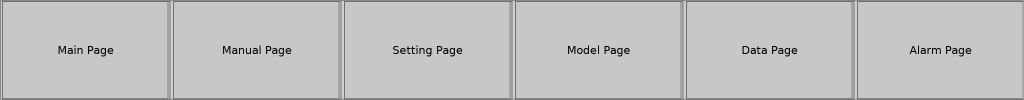
VISUALIZATION LowerBar  // 1024x100
    Button (2,1 168x99), "Main Page", colour toggle: gvl_hmi.bMainScreen
        OnMouseClick: execute { gvl_hmi.iMainFrame := 0; }
    Button (173,1 168x99), "Manual Page", colour toggle: gvl_hmi.bManualScreen
        OnMouseClick: execute { gvl_hmi.iMainFrame := 1; }
    Button (344,1 168x99), "Setting Page", colour toggle: gvl_hmi.bSettingScreen
        OnMouseClick: execute { gvl_hmi.iMainFrame := 2; }
    Button (515,1 168x99), "Model Page", colour toggle: gvl_hmi.bModelScreen
        OnMouseClick: execute { gvl_hmi.iMainFrame := 3; }
    Button (686,1 168x99), "Data Page", colour toggle: gvl_hmi.bDataScreen
        OnMouseClick: execute { gvl_hmi.iMainFrame := 4; }
    Button (857,1 168x99), "Alarm Page", colour toggle: gvl_hmi.bAlarmScreen
        OnMouseClick: execute { gvl_hmi.iMainFrame := 5; }
END_VISUALIZATION

(* stored: Version 1.1.0.1
   Visu LowerBar: Id {e0ed94dc-2c48-4488-bf7a-f81f7695db5c} *)
